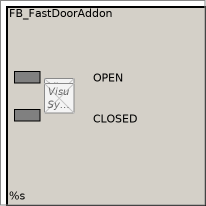
VISUALIZATION V_FastDoorAddon  // 206x206
VAR_IN_OUT
	fbFunction 	: FB_FastDoorAddon;
END_VAR
    Rectangle (6,6 200x200)
    Rectangle (6,186 200x20), "%s", text variable: fbFunction.ConfigFunction.FunctionName
    Label (6,6 200x15), "FB_FastDoorAddon"
    Rectangle (14,109 26x12), tooltip "Door lift sensor", colour toggle: fbFunction.HW_Inputs.Closed
    Rectangle (14,71 26x12), tooltip "Door up sensor", colour toggle: fbFunction.HW_Inputs.Open
    Image (44,78 30x30), tooltip "Door moving up", invisible if: NOT fbFunction.HW_Outputs.OpenDoor, image: VisuSymbols.Symbols.ArrowBoldUp
    Image (44,83 30x30), tooltip "Door moving down", invisible if: NOT fbFunction.HW_Outputs.CloseDoor, image: VisuSymbols.Symbols.ArrowBoldDown
    Rectangle (90,68 60x20), "OPEN", tooltip "Door open", text variable: fbFunction.ConfigFunction.FunctionName, invisible if: NOT fbFunction.HW_Inputs.Open
    Rectangle (90,109 60x20), "CLOSED", tooltip "Door closed", text variable: fbFunction.ConfigFunction.FunctionName, invisible if: NOT fbFunction.HW_Inputs.Closed
END_VISUALIZATION

(* stored: Version 1.1.0.1, ProductVersion 3.1.4024.9
   Visu V_FastDoorAddon: Id {86200875-df8a-4fa6-a275-f847d9ff16a7} *)
